
// ===== library types =====

TYPE "udtError_MQTT"
   STRUCT
      ConSendErr : Bool;   // Connect send error
      ConSendTO : Bool;   // Connect send timeout
      ConAckRcvErr : Bool;   // Connack receive error
      ConAckTO : Bool;   // Connack timeout
      ConAckIncReply : Bool;   // Conack incorrect reply (header)
      ConAckIncLen : Bool;   // Conack incorrect remaining length
      ConAckUnacProt : Bool;   // Conack unacceptable protocol version (0x01)
      ConAckIdRej : Bool;   // Conack ID rejected (0x02)
      ConAckSerUn : Bool;   // Conack server unavailable (0x03)
      ConAckUserPass : Bool;   // Conack incorerct user/password (0x04)
      ConAckNotAut : Bool;   // Conack not authorized (0x05)
      ConAckUnknown : Bool;   // Conack unknow erro code (>0x05)
      PubSendErr : Bool;   // Publish send error
      PubSendTO : Bool;   // Publish send timeout
      PubAckRcvErr : Bool;   // Puback receive error
      PubAckTO : Bool;   // Puback receive timeout
      PubAckIncReply : Bool;   // Puback incorerct reply (header)
      PubAckIncLen : Bool;   // Puback incorrect remaining length
      PubAckPacketID : Bool;   // Puback incorrect Packet ID
      SubSendErr : Bool;   // Subscribe send error
      SubSendTimeout : Bool;   // Subscribe send timeout
      SubAckIncReply : Bool;   // Suback incorrect reply
      SubAckPacketID : Bool;   // Suback incorrect Packet ID
      SubAckRcvErr : Bool;   // Suback receive error
      SubAckTO : Bool;   // Suback receive timeout
      SubTopicNotFound : Bool;   // Message sent to PLC, but not subscribed to topic
      SubSendPubAckErr : Bool;   // Error sending pub ack message
      SubSendPubAckTO : Bool;   // Send pub ack timeout
      TcpErr : Bool;   // TCP connection failed
      TcpTO : Bool;   // TCP connection timeout
      QueueOverflow : Bool;   // Queue overlow
   END_STRUCT;
END_TYPE

TYPE "udtMQTT_PublishMessage"
   STRUCT
      iStatus : Int;   // 0 - Disabled,10 - Ready to Send
      iQoS : Int;
      sTopic : String;
      byValue : Array[0..100] of Byte;
      iMessageLength : DInt;
   END_STRUCT;
END_TYPE

TYPE "udtMQTT_PublishMessageBuffer"
   STRUCT
      iIndexWrite : Int;
      iIndexMax : Int := 50;
      bErrorOverfill : Bool;
      Message : Array[1..10] of "udtMQTT_PublishMessage";
   END_STRUCT;
END_TYPE

TYPE "udtMQTT_SubscribeMessage"
   STRUCT
      iStatus : Int;   // 0 - Disabled, 10 - Ready to subscribe, 20 - subscribed, 30 - New data
      iQoS : Int;
      sTopic : String[75];
      byValue : Array[0..75] of Byte;
      iMessageLength : Int;
   END_STRUCT;
END_TYPE

TYPE "udtMQTT_SubcribeMessageBuffer"
   STRUCT
      Message : Array[1..20] of "udtMQTT_SubscribeMessage";
   END_STRUCT;
END_TYPE

FUNCTION_BLOCK "fbMQTT_V2"   // FB19, SCL
{ S7_Optimized_Access := 'TRUE' }
VERSION : 0.1
   VAR_INPUT
      sInClientID : String;   // Client ID, 23 char max
      sInUserName : String;
      sInPassword : String;
      bInCleanSession : Bool;   // 0=Reuse prev session; 1=Discard prev sessions and start new one
      bInResetError : Bool;
   END_VAR
   VAR_OUTPUT
      bOutError : Bool;
   END_VAR
   VAR_IN_OUT
      ERROR_MQTT : "udtError_MQTT";
      TCON_Param : TCON_Param;
   END_VAR
   VAR
      iStatePublish : Int;
      iStateSubscribe : Int;
      iStateTCP_Receive : Int;
      iSelQueueIndexPublish : Int;
      iPublishIndex : Int;
      uiSendLen : UInt;
      udiReceiveLen : UDInt;
      uiPubPacketID : UInt;
      bPubInProgress : Bool;
      iSubscribeIndex : Int;
      uiSubPacketID : UInt;
      iSubMessageIndex : Int;
      bSubInProgress : Bool;
      bSubReceiveInProgress : Bool;
      iSubReceivedQoS : Int;
      iReceivedTopicLength : Int;
      sReceivedTopic : String;
      iTopicIndex : Int;
      bConAckReceived : Bool;
      bPubAckReceived : Bool;
      bSubAckReceived : Bool;
      bPublishReceived : Bool;
      iPayloadStartIndex : Int;
      iEndOfPayloadIndex : Int;
      byData : Array[1..200] of Byte;   // Max: id+user+password+buffer
      byDataNewMessage : Array[1..300] of Byte;
      fbTCON : TCON;
      fbTDISCON : TDISCON;
      fbTSEND : TSEND;
      fbTRCV : TRCV;
      TON_TimeoutPub : TON_TIME;
      TON_TimeoutSub : TON_TIME;
      TON_ReceiveDataComplete : TON_TIME;
      TON_DelaySubscribe : TON_TIME;   // To space out traffic, wait 5 seconds after MQTT connection to subscribe
      iNewDataIndex : Int := 1;
      bNewDataReceived : Bool;
      bTCP_Connected : Bool;
      bMQTT_Connected : Bool;
      iLen : Int;
      iStatePrevPub : Int;
      bStateTransitionPub : Bool;
      udiSetReceiveLen : UDInt;
      wTemp : Word;
      wTemp2 : Word;
      wTemp3 : Word;
      wTemp4 : Word;
      byMSB : Byte;
      byLSB : Byte;
      iStatePrevSub : Int;
      bStateTransitionSub : Bool;
      bReceiveMessageComplete : Bool;
      iReceiveMessageLength : Int;
      iReceiveLengthCalcIndex : Int;
      iErrIndex : Int := 1;
   END_VAR
   VAR_TEMP
      i : Int;
      j : Int;
      iStartingIndex : Int;
      iTemp : Int;
      byTemp : Byte;
      uiTemp : UInt;
      uiTopicLen : UInt;
      multiplier : Int;
      byTopic : Array[1..500] of Byte;
      byReceivedPayload : Array[1..500] of Byte;
      iLowerByte : Int;
      iHigherByte : Int;
      sSearchString : String;
      bTopicNotFound : Bool;
   END_VAR
   VAR CONSTANT
      ciPublishQueueSize : Int := 10;
      ciPubIdle : Int := 10;
      ciPubError : Int := 999;
      ciEstablishTCP : Int := 100;
      ciPubConnect : Int := 20;
      ciPubConnectSend : Int := 30;
      ciPubWaitConnack : Int := 40;
      ciPubPublish : Int := 50;
      ciPubSend : Int := 60;
      ciPubWaitPubAck : Int := 70;
      ciPubRestart : Int := -1;
      ciSubQueueSize : Int := 20;
      ciSubIdle : Int := 10;
      ciSubError : Int := 999;
      ciSubWaitTCP : Int := 20;
      ciSubSubscribe : Int := 30;
      ciSubSendSubscribe : Int := 40;
      ciSubWaitSuback : Int := 50;
      ciSubDataReceived : Int := 60;
      ciSubSendPubAck : Int := 70;
      ciRecIdle : Int := 10;
      ciRecDataReceived : Int := 20;
      ciRecParseData : Int := 30;
      ciRecConAck : Int := 40;
      ciRecPubAck : Int := 50;
      ciRecSubAck : Int := 60;
      ciRecPubReceived : Int := 70;
   END_VAR
BEGIN
   //Publish state machine
   //Test comment
   #iStatePrevPub := #iStatePublish;
   CASE #iStatePublish OF
       #ciPubIdle:
           // Update max queue index
           "dbMQTT_MessageBuffer".OutgoingMessages.iIndexMax := #ciPublishQueueSize;

           //connect by default
           IF NOT #bTCP_Connected THEN
               #iStatePublish := #ciEstablishTCP;
           END_IF;

           IF #bTCP_Connected AND NOT #bMQTT_Connected THEN
               #iStatePublish := #ciPubConnect;
           END_IF;


           // Already select element to send?
           IF #iSelQueueIndexPublish > 0 THEN
               IF #bTCP_Connected AND #bMQTT_Connected AND #iStateSubscribe = #ciSubIdle THEN
                   //Only publish if subscribe state machine is also idle
                   #iStatePublish := #ciPubPublish;
               END_IF;
           ELSE
               // Find element in the queue to send
               FOR #i := 1 TO "dbMQTT_MessageBuffer".OutgoingMessages.iIndexMax DO
                   // Check if element is ready in the queue
                   IF ("dbMQTT_MessageBuffer".OutgoingMessages.Message[#i].iStatus = "ciReadyToPublish") THEN
                       #iSelQueueIndexPublish := #i;
                       EXIT;
                   END_IF;
               END_FOR;
           END_IF;

       #ciPubConnect: // Send connect message
           ////////////////////////////////////
           // Create connect message
           ////////////////////////////////////

           //********* Configure Fixed Header ***********//
           #iPublishIndex := 1;
           #byData[#iPublishIndex] := 2#00010000;   // Packet type 0x1; Flags 0x0 (reserved)
           #iPublishIndex := #iPublishIndex + 1;

           //Reset all subscriptions
           FOR #i := 1 TO 20 BY 1 DO
               "dbMQTT_MessageBuffer".IncomingMessages.Message[#i].iStatus := "ciSubDisabled";
           END_FOR;

           // Calculate remaining length (see MQTT doc)
           #iLen := 12 + LEN(#sInClientID);
           IF LEN(#sInUserName) > 0 THEN
               #iLen := #iLen + LEN(#sInUserName) + 2;
           END_IF;
           IF LEN(#sInPassword) > 0 THEN
               #iLen := #iLen + LEN(#sInPassword) + 2;
           END_IF;
           REPEAT
               #byTemp := INT_TO_BYTE(#iLen MOD 128);
               #iLen := #iLen / 128;
               // if there are more data to encode, set the top bit of this byte 286
               IF #iLen > 0 THEN
                   #byTemp := #byTemp OR 128;
               END_IF;
               #byData[#iPublishIndex] := #byTemp;
               #iPublishIndex := #iPublishIndex + 1;
           UNTIL #iLen <= 0 END_REPEAT;

           //********* Variable Header ***********//
           #byData[#iPublishIndex] := 16#00;    // Length MSB
           #iPublishIndex := #iPublishIndex + 1;
           #byData[#iPublishIndex] := 16#04;    // Length LSB
           #iPublishIndex := #iPublishIndex + 1;
           #byData[#iPublishIndex] := CHAR_TO_BYTE('M');
           #iPublishIndex := #iPublishIndex + 1;
           #byData[#iPublishIndex] := CHAR_TO_BYTE('Q');
           #iPublishIndex := #iPublishIndex + 1;
           #byData[#iPublishIndex] := CHAR_TO_BYTE('T');
           #iPublishIndex := #iPublishIndex + 1;
           #byData[#iPublishIndex] := CHAR_TO_BYTE('T');
           #iPublishIndex := #iPublishIndex + 1;
           #byData[#iPublishIndex] := 16#04;     // Protocol level 0x04
           #iPublishIndex := #iPublishIndex + 1;

           // Build connect flags, ignoring will message
           #byData[#iPublishIndex] := 16#00;
           IF LEN(#sInUserName) > 0 THEN
               #byData[#iPublishIndex] := #byData[#iPublishIndex] OR 2#10000000;
           END_IF;
           IF LEN(#sInPassword) > 0 THEN
               #byData[#iPublishIndex] := #byData[#iPublishIndex] OR 2#01000000;
           END_IF;
           IF #bInCleanSession THEN
               #byData[#iPublishIndex] := #byData[#iPublishIndex] OR 2#00000010;
           END_IF;
           #iPublishIndex := #iPublishIndex + 1;
           #byData[#iPublishIndex] := 16#0E;  // Keepalive MSB, in seconds
           #iPublishIndex := #iPublishIndex + 1;
           #byData[#iPublishIndex] := 16#10;  // Keepalive LSB, in seconds
           #iPublishIndex := #iPublishIndex + 1;

           // Payload - client ID
           #iLen := LEN(#sInClientID);
           #byData[#iPublishIndex] := WORD_TO_BYTE(SHR(IN := INT_TO_WORD(#iLen), N := 8));   // String lenght MSB
           #iPublishIndex := #iPublishIndex + 1;
           #byData[#iPublishIndex] := WORD_TO_BYTE(INT_TO_WORD(#iLen) AND 16#00FF);   // String lenght LSB            
           #iPublishIndex := #iPublishIndex + 1;
           FOR #i := 1 TO #iLen DO
               #byData[#iPublishIndex] := CHAR_TO_BYTE(#sInClientID[#i]);
               #iPublishIndex := #iPublishIndex + 1;
           END_FOR;

           // Payload - User name
           IF LEN(#sInUserName) > 0 THEN
               #iLen := LEN(#sInUserName);
               #byData[#iPublishIndex] := WORD_TO_BYTE(SHR(IN := INT_TO_WORD(#iLen), N := 8));   // String lenght MSB
               #iPublishIndex := #iPublishIndex + 1;
               #byData[#iPublishIndex] := WORD_TO_BYTE(INT_TO_WORD(#iLen) AND 16#00FF);   // String lenght LSB            
               #iPublishIndex := #iPublishIndex + 1;
               FOR #i := 1 TO #iLen DO
                   #byData[#iPublishIndex] := CHAR_TO_BYTE(#sInUserName[#i]);
                   #iPublishIndex := #iPublishIndex + 1;
               END_FOR;
           END_IF;

           // Payload - password
           IF LEN(#sInPassword) > 0 THEN
               #iLen := LEN(#sInPassword);
               #byData[#iPublishIndex] := WORD_TO_BYTE(SHR(IN := INT_TO_WORD(#iLen), N := 8));   // String lenght MSB
               #iPublishIndex := #iPublishIndex + 1;
               #byData[#iPublishIndex] := WORD_TO_BYTE(INT_TO_WORD(#iLen) AND 16#00FF);   // String lenght LSB            
               #iPublishIndex := #iPublishIndex + 1;
               FOR #i := 1 TO #iLen DO
                   #byData[#iPublishIndex] := CHAR_TO_BYTE(#sInPassword[#i]);
                   #iPublishIndex := #iPublishIndex + 1;
               END_FOR;
           END_IF;

           //********* Send Packet ***********//
           #uiSendLen := INT_TO_UINT(#iPublishIndex - 1);   // Update packet length
           #iStatePublish := #ciPubConnectSend;  // Send packet packet

       #ciPubConnectSend:
           IF #fbTSEND.DONE THEN
               // All good. Receive conack message
               // We know exactly the conack message size
               #udiReceiveLen := 4;
               #iStatePublish := #ciPubWaitConnack;
           ELSIF #fbTSEND.ERROR THEN
               // Sending error
               #ERROR_MQTT.ConSendErr := true;
               #iStatePublish := #ciPubError;
           ELSIF #TON_TimeoutPub.Q THEN
               #ERROR_MQTT.ConSendTO := true;
               #iStatePublish := #ciPubError;
           END_IF;

       #ciPubWaitConnack:
           IF #bConAckReceived THEN
               //Reset received flag
               #bConAckReceived := FALSE;
               // Parse received data
               // We know that we got an expected length
               // Header should be 0x20
               IF #byDataNewMessage[1] <> 16#20 THEN
                   #ERROR_MQTT.ConAckIncReply := true;
                   #iStatePublish := #ciPubError;
                   // Remaining lenght should be 2
               ELSIF #byDataNewMessage[2] <> 2 THEN
                   #ERROR_MQTT.ConAckIncLen := true;
                   #iStatePublish := #ciPubError;
                   // TODO: Parse SP flag?
                   // Return code should be 0    
               ELSIF #byDataNewMessage[4] <> 0 THEN
                   // Parse error code
                   IF #byDataNewMessage[4] = 1 THEN
                       #ERROR_MQTT.ConAckUnacProt := TRUE;
                   ELSIF #byDataNewMessage[4] = 2 THEN
                       #ERROR_MQTT.ConAckIdRej := TRUE;
                   ELSIF #byDataNewMessage[4] = 3 THEN
                       #ERROR_MQTT.ConAckSerUn := TRUE;
                   ELSIF #byDataNewMessage[4] = 4 THEN
                       #ERROR_MQTT.ConAckUserPass := TRUE;
                   ELSIF #byDataNewMessage[4] = 5 THEN
                       #ERROR_MQTT.ConAckNotAut := TRUE;
                   ELSE
                       #ERROR_MQTT.ConAckUnknown := TRUE;
                   END_IF;
                   #iStatePublish := #ciPubError;
               ELSE
                   // All good
                   #bMQTT_Connected := true;
                   #iStatePublish := #ciPubIdle;
               END_IF;
           (*ELSIF #fbTRCV.ERROR THEN
               // Receive error
               #ERROR_MQTT.ConAckRcvErr := true;
               "dbTestingJJC".wDisError := #fbTRCV.STATUS;
               #iStatePublish := #ciPubError;*)
           ELSIF #TON_TimeoutPub.Q THEN
               #ERROR_MQTT.ConAckTO := true;
               #iStatePublish := #ciPubError;
           END_IF;

       #ciPubPublish:
           ////////////////////////////////////
           // Create publish message
           ////////////////////////////////////

           //********* Configure Fixed Header ***********//
           #iPublishIndex := 1;
           #byData[#iPublishIndex] := 2#00110000;   // Packet type 0x3;
           IF #bPubInProgress THEN
               #byData[#iPublishIndex] := #byData[#iPublishIndex] OR 2#00001000; // DUP flag. Re-delivery attempt
           ELSE
               // New send attempt - Increment Packet ID
               #uiPubPacketID := #uiPubPacketID + 1;
           END_IF;
           // QoS flag, assuming 0 by default
           IF "dbMQTT_MessageBuffer".OutgoingMessages.Message[#iSelQueueIndexPublish].iQoS = 1 THEN
               #byData[#iPublishIndex] := #byData[#iPublishIndex] OR 2#00000010; // QoS flag
           END_IF;
           //TODO: QoS 2 is not currently implemented by adafruit
           // TODO: Ignoring retain flag for now
           #iPublishIndex := #iPublishIndex + 1;

           // Calculate remaining length (see MQTT doc)
           // No lenght for the payload
           #iLen := LEN("dbMQTT_MessageBuffer".OutgoingMessages.Message[#iSelQueueIndexPublish].sTopic) + 2 + DINT_TO_INT("dbMQTT_MessageBuffer".OutgoingMessages.Message[#iSelQueueIndexPublish].iMessageLength);
           IF "dbMQTT_MessageBuffer".OutgoingMessages.Message[#iSelQueueIndexPublish].iQoS > 0 THEN
               // Adding packet ID for QoS 1 and 2
               #iLen := #iLen + 2;
           END_IF;
           REPEAT
               #byTemp := INT_TO_BYTE(#iLen MOD 128);
               #iLen := #iLen / 128;
               // if there are more data to encode, set the top bit of this byte 286
               IF #iLen > 0 THEN
                   #byTemp := #byTemp OR 128;
               END_IF;
               #byData[#iPublishIndex] := #byTemp;
               #iPublishIndex := #iPublishIndex + 1;
           UNTIL #iLen <= 0 END_REPEAT;

           //********* Variable Header ***********//
           // Topic name
           #iLen := LEN("dbMQTT_MessageBuffer".OutgoingMessages.Message[#iSelQueueIndexPublish].sTopic);
           #byData[#iPublishIndex] := WORD_TO_BYTE(SHR(IN := INT_TO_WORD(#iLen), N := 8));   // String lenght MSB
           #iPublishIndex := #iPublishIndex + 1;
           #byData[#iPublishIndex] := WORD_TO_BYTE(INT_TO_WORD(#iLen) AND 16#00FF);   // String lenght LSB
           #iPublishIndex := #iPublishIndex + 1;
           FOR #i := 1 TO #iLen DO
               #byData[#iPublishIndex] := CHAR_TO_BYTE("dbMQTT_MessageBuffer".OutgoingMessages.Message[#iSelQueueIndexPublish].sTopic[#i]);
               #iPublishIndex := #iPublishIndex + 1;
           END_FOR;
           // packet ID
           IF "dbMQTT_MessageBuffer".OutgoingMessages.Message[#iSelQueueIndexPublish].iQoS > 0 THEN
               #byData[#iPublishIndex] := WORD_TO_BYTE(SHR(IN := UINT_TO_WORD(#uiPubPacketID), N := 8));   // Packet ID MSB
               #iPublishIndex := #iPublishIndex + 1;
               #byData[#iPublishIndex] := WORD_TO_BYTE(UINT_TO_WORD(#uiPubPacketID) AND 16#00FF);   // PacketID LSB
               #iPublishIndex := #iPublishIndex + 1;
           END_IF;

           //********* Payload ***********//
           // The exact data format is not defined in the MQTT spec
           // Assuming strings, without string length
           // According to the spec, server should calcualte the lenght of the payload
           #iLen := DINT_TO_INT("dbMQTT_MessageBuffer".OutgoingMessages.Message[#iSelQueueIndexPublish].iMessageLength);
           FOR #i := 0 TO #iLen - 1 DO
               #byData[#iPublishIndex] := "dbMQTT_MessageBuffer".OutgoingMessages.Message[#iSelQueueIndexPublish].byValue[#i];
               #iPublishIndex := #iPublishIndex + 1;
           END_FOR;

           // Send message
           #bPubInProgress := true;
           #uiSendLen := INT_TO_UINT(#iPublishIndex - 1);   // Update packet length
           #iStatePublish := #ciPubSend;

       #ciPubSend:
           IF #fbTSEND.DONE THEN
               // QoS=1: Should receive puback message
               IF "dbMQTT_MessageBuffer".OutgoingMessages.Message[#iSelQueueIndexPublish].iQoS = 1 THEN
                   #udiReceiveLen := 4;    // Wes should receive exactly 4 bytes
                   #iStatePublish := #ciPubWaitPubAck;
               ELSE
                   // QoS=0; No response from the server
                   // Remove message from the queue
                   "dbMQTT_MessageBuffer".OutgoingMessages.Message[#iSelQueueIndexPublish].iStatus := "ciDisablePublish";
                   #iSelQueueIndexPublish := 0;
                   #bPubInProgress := false;
                   #iStatePublish := #ciPubIdle;
               END_IF;
               // TODO: Handle QoS 2?
           ELSIF #fbTSEND.ERROR THEN
               // Send error
               #ERROR_MQTT.PubSendErr := true;
               #iStatePublish := #ciPubError;
           ELSIF #TON_TimeoutPub.Q THEN
               #ERROR_MQTT.PubSendTO := true;
               #iStatePublish := #ciPubError;
           END_IF;

       #ciEstablishTCP:
           // Wait for done or error flag
           IF #fbTCON.DONE THEN
               // TCP connection established 
               #bTCP_Connected := true;
               #bMQTT_Connected := false;
               #iStatePublish := #ciPubConnect;
           ELSIF #fbTCON.ERROR THEN
               // Connection failed
               #ERROR_MQTT.TcpErr := true;
               IF #fbTCON.STATUS = 16#80A3 THEN
                   #TCON_Param.ID := #TCON_Param.ID + 1;
               END_IF;
               IF #TCON_Param.ID > 9 THEN
                   #TCON_Param.ID := 1;
               END_IF;
               #iStatePublish := #ciPubError;
           ELSIF #TON_TimeoutPub.Q THEN
               #ERROR_MQTT.TcpTO := true;
               #iStatePublish := #ciPubError;
           END_IF;

       #ciPubWaitPubAck:
           IF #bPubAckReceived THEN
               #bPubAckReceived := false;
               // Parse received data
               // We know that we got an expected length
               // Header should be 0x40
               IF #byDataNewMessage[2] <> 16#02 THEN
                   // Wrong pub ack remaining lenght
                   // TODO pub ack length error
                   #iStatePublish := #ciPubError;
               ELSE
                   // Variable header = message id
                   #uiTemp := WORD_TO_UINT(SHL(IN := BYTE_TO_WORD(#byDataNewMessage[3]), N := 8) + BYTE_TO_WORD(#byDataNewMessage[4]));
                   IF #uiTemp <> #uiPubPacketID THEN
                       // Incorerct packet ID
                       #ERROR_MQTT.PubAckPacketID := TRUE;
                       #iStatePublish := #ciPubError;
                   ELSE
                       // All good. Reset queue and restart
                       "dbMQTT_MessageBuffer".OutgoingMessages.Message[#iSelQueueIndexPublish].iStatus := "ciDisablePublish";
                       #iSelQueueIndexPublish := 0;
                       #bPubInProgress := false;
                       #iStatePublish := #ciPubIdle;
                   END_IF;
               END_IF;
           ELSIF #fbTRCV.ERROR THEN
               // Receive error
               #ERROR_MQTT.PubAckRcvErr := TRUE;
               #iStatePublish := #ciPubError;
           ELSIF #TON_TimeoutPub.Q THEN
               #ERROR_MQTT.PubAckTO := true;
               #iStatePublish := #ciPubError;
           END_IF;

       #ciPubError:
           // Reset TCP connection
           #bMQTT_Connected := false;
           #bTCP_Connected := false;
           IF #fbTDISCON.DONE THEN
               #iStatePublish := #ciPubRestart;
           ELSIF #TON_TimeoutPub.Q THEN
               // Already wait for timeout, just jump to idle
               #iStatePublish := #ciPubIdle;
               #iNewDataIndex := 1;
           END_IF;

       #ciPubRestart:
           // Wait before restarting after the error
           IF #TON_TimeoutPub.Q THEN
               // Restart from IDLE
               #iStatePublish := #ciPubIdle;
               #iNewDataIndex := 1;
           END_IF;

       ELSE
           #iStatePublish := #ciPubIdle;

   END_CASE;

   // Timeoout timer
   #bStateTransitionPub := #iStatePublish <> #iStatePrevPub;
   #TON_TimeoutPub(IN := ((NOT #bStateTransitionPub) AND (#iStatePublish <> #ciPubIdle) AND #iStateSubscribe = #ciSubIdle), PT := T#20S);

   //subscribe state machine
   #iStatePrevSub := #iStateSubscribe;
   CASE #iStateSubscribe OF
       #ciSubIdle:
           #bSubInProgress := false;
           #bSubReceiveInProgress := false;
           //Wait until TCP and MQTT connected and publish is idle
           IF #TON_DelaySubscribe.Q AND #iStatePublish = #ciPubIdle  THEN
               //check if any new data has arrived
               IF #bPublishReceived THEN
                   //Reset flag
                   #bPublishReceived := false;
                   //if data has arrived, move to data received state
                   #iStateSubscribe := #ciSubDataReceived;
                   //Set flag to prevent sending other messages out
                   #bSubReceiveInProgress := true;
               END_IF;

               //check for any unsubscribed topics
               IF NOT #bSubReceiveInProgress THEN
                   FOR #i := 1 TO #ciSubQueueSize BY 1 DO
                       IF "dbMQTT_MessageBuffer".IncomingMessages.Message[#i].iStatus = "ciSubReadyToSub" THEN
                           //If unsubscribed topic found, move to sub state and stop looking for new topics
                           #iStateSubscribe := #ciSubSubscribe;
                           #iSubscribeIndex := #i;
                           #bSubInProgress := TRUE;
                           EXIT;
                       END_IF;
                   END_FOR;
               END_IF;
           END_IF;

       #ciSubSubscribe:
           //create subscribe MQTT packet
           #i := 1;
           #iSubMessageIndex := 1;
           #byData[#iSubMessageIndex] := 2#10000010;   // Packet type 0x8; Flags 0x0 (reserved)
           #iSubMessageIndex := #iSubMessageIndex + 1;

           // Calculate remaining length (see MQTT doc)
           // packet identifier (2) + topic length (2) + length of topic + QoS (1)
           #iLen := LEN("dbMQTT_MessageBuffer".IncomingMessages.Message[#iSubscribeIndex].sTopic) + 5;
           //Create encoding for packet length
           REPEAT
               #byTemp := INT_TO_BYTE(#iLen MOD 128);
               #iLen := #iLen / 128;
               // if there are more data to encode, set the top bit of this byte 286
               IF #iLen > 0 THEN
                   #byTemp := #byTemp OR 128;
               END_IF;
               #byData[#iSubMessageIndex] := #byTemp;
               #iSubMessageIndex := #iSubMessageIndex + 1;
           UNTIL #iLen <= 0 END_REPEAT;
           //increment packet ID and encode into variable header
           #uiSubPacketID := #uiSubPacketID + 1;
           #byData[#iSubMessageIndex] := WORD_TO_BYTE(SHR(IN := UINT_TO_WORD(#uiSubPacketID), N := 8));   // Packet ID MSB
           #iSubMessageIndex := #iSubMessageIndex + 1;
           #byData[#iSubMessageIndex] := WORD_TO_BYTE(UINT_TO_WORD(#uiSubPacketID) AND 16#00FF);   // PacketID LSB
           #iSubMessageIndex := #iSubMessageIndex + 1;

           //build payload
           //Only 1 topic. 2 bytes for length, topic, 1 byte for QoS
           //Length
           #uiTopicLen := INT_TO_UINT(LEN("dbMQTT_MessageBuffer".IncomingMessages.Message[#iSubscribeIndex].sTopic));
           #byData[#iSubMessageIndex] := WORD_TO_BYTE(SHR(IN := UINT_TO_WORD(#uiTopicLen), N := 8));   // Packet ID MSB
           #iSubMessageIndex := #iSubMessageIndex + 1;
           #byData[#iSubMessageIndex] := WORD_TO_BYTE(UINT_TO_WORD(#uiTopicLen) AND 16#00FF);   // PacketID LSB
           #iSubMessageIndex := #iSubMessageIndex + 1;
           // Topic name
           #iLen := LEN("dbMQTT_MessageBuffer".IncomingMessages.Message[#iSubscribeIndex].sTopic);
           FOR #i := 1 TO #iLen DO
               #byData[#iSubMessageIndex] := CHAR_TO_BYTE("dbMQTT_MessageBuffer".IncomingMessages.Message[#iSubscribeIndex].sTopic[#i]);
               #iSubMessageIndex := #iSubMessageIndex + 1;

           END_FOR;
           //QoS
           IF "dbMQTT_MessageBuffer".IncomingMessages.Message[#iSubscribeIndex].iQoS = 1 THEN
               #byData[#iSubMessageIndex] := 2#00000001;
           ELSE
               #byData[#iSubMessageIndex] := 2#00000000;
           END_IF;
           #uiSendLen := INT_TO_UINT(#iSubMessageIndex);
           #iStateSubscribe := #ciSubSendSubscribe;

       #ciSubSendSubscribe:
           IF #fbTSEND.DONE THEN

               #iStateSubscribe := #ciSubWaitSuback;
               IF "dbMQTT_MessageBuffer".IncomingMessages.Message[#iSubscribeIndex].iQoS = 0 THEN
                   #udiReceiveLen := 5;    // Wes should receive exactly 4 bytes
                   #iStateSubscribe := #ciSubWaitSuback;
               END_IF;
           ELSIF #fbTSEND.ERROR THEN
               // Send error
               #ERROR_MQTT.PubSendErr := true;
               #iStateSubscribe := #ciPubError;
           ELSIF #TON_TimeoutSub.Q THEN
               #ERROR_MQTT.PubSendTO := true;
               #iStateSubscribe := #ciPubError;
           END_IF;

       #ciSubWaitSuback:
           //validate packet received. Should have same packet ID
           //
           IF #bSubAckReceived THEN
               #bSubAckReceived := false;
               // Parse received data
               // We know that we got an expected length
               // Header should be 0x40

               // Variable header = message id
               #uiTemp := WORD_TO_UINT(SHL(IN := BYTE_TO_WORD(#byDataNewMessage[3]), N := 8) + BYTE_TO_WORD(#byDataNewMessage[4]));

               IF #uiTemp <> #uiSubPacketID THEN
                   // Incorerct packet ID
                   #ERROR_MQTT.SubAckPacketID := TRUE;
                   #iStateSubscribe := #ciSubError;
                   //TODO also check QoS?
               ELSE
                   // All good. Reset queue and restart

                   "dbMQTT_MessageBuffer".IncomingMessages.Message[#iSubscribeIndex].iStatus := "ciSubSubscribed";
                   #iStateSubscribe := #ciSubIdle;
               END_IF;
           (* ELSIF #fbTRCV.ERROR THEN
               // Receive error
               #ERROR_MQTT.SubAckRcvErr := TRUE;
               #iStateSubscribe := #ciSubError; *)
           ELSIF #TON_TimeoutSub.Q THEN
               #ERROR_MQTT.SubAckTO := true;
               #iStateSubscribe := #ciSubError;
           END_IF;


       #ciSubDataReceived:
           //reset flag
           #bSubReceiveInProgress := false;
           //find QoS
           #iSubMessageIndex := 1;
           #iSubReceivedQoS := 0;
           //TODO handling for QoS 2
           IF (#byDataNewMessage[#iSubMessageIndex] AND 2#00000010) = 2#00000010 THEN
               #iSubReceivedQoS := 1;
           END_IF;

           //calculate message length
           #multiplier := 1;
           #iLen := 0;
           #iSubMessageIndex := 2;
           REPEAT

               #byTemp := #byDataNewMessage[#iSubMessageIndex];
               #iLen := #iLen + (#byTemp AND 127) * #multiplier;
               #multiplier := #multiplier * 128;
               //TODO implement exception for length error

               #iSubMessageIndex := #iSubMessageIndex + 1;
           UNTIL ((#byTemp AND 128) = 0) END_REPEAT;

           //find end index of message
           #iEndOfPayloadIndex := #iLen + #iSubMessageIndex - 1;

           //find topic name
           //find topic length
           #wTemp := 16#0000;
           #wTemp2 := 16#0000;
           #wTemp := #wTemp OR #byDataNewMessage[#iSubMessageIndex];
           #iSubMessageIndex := #iSubMessageIndex + 1;
           #wTemp2 := #byDataNewMessage[#iSubMessageIndex];
           #wTemp3 := SHL(IN := #wTemp, N := 8);
           #wTemp4 := #wTemp OR #wTemp2;
           #iReceivedTopicLength := WORD_TO_INT(IN := #wTemp4);
           #iSubMessageIndex := #iSubMessageIndex + 1;
           #iStartingIndex := #iSubMessageIndex;
           #j := 1;
           FOR #i := #iStartingIndex TO #iStartingIndex + #iReceivedTopicLength BY 1 DO
               #byTopic[#j] := #byDataNewMessage[#iSubMessageIndex];
               #j := #j + 1;
               #iSubMessageIndex := #iSubMessageIndex + 1;
           END_FOR;

           Chars_TO_Strg(Chars:=#byTopic, pChars:=0, Cnt:=INT_TO_UINT(#iReceivedTopicLength), Strg=>#sReceivedTopic);
           //find index of topic
           #bTopicNotFound := TRUE;
           FOR #i := 1 TO #ciSubQueueSize BY 1 DO

               IF ("dbMQTT_MessageBuffer".IncomingMessages.Message[#i].sTopic = #sReceivedTopic) THEN
                   #iTopicIndex := #i;
                   #bTopicNotFound := FALSE;
                   EXIT;
               END_IF;
           END_FOR;

           //Throw error if topic not found
           IF #bTopicNotFound THEN
               #ERROR_MQTT.SubTopicNotFound := TRUE;
               #iStatePrevSub := #ciSubError;
           END_IF;

           //Depending on QoS go to idle or send PubAck reply
           IF (#iSubReceivedQoS = 0) THEN
               #iStateSubscribe := #ciSubIdle;
           ELSIF (#iSubReceivedQoS = 1) THEN

               //Find packet ID
               #byLSB := #byDataNewMessage[#iSubMessageIndex];
               #iSubMessageIndex := #iSubMessageIndex + 1;
               #byMSB := #byDataNewMessage[#iSubMessageIndex];

               //build reply message
               //Control packet 16#40
               #byData[1] := 16#40;
               //remaining length is 2
               #byData[2] := 16#02;
               //add packet id
               #byData[3] := #byMSB;
               #byData[4] := #byLSB;
               #uiSendLen := 4;

               #iStateSubscribe := #ciSubSendPubAck;
           END_IF;

           //get message
           IF NOT #bTopicNotFound THEN
               #iPayloadStartIndex := #iSubMessageIndex;
               #j := 0;
               FOR #i := #iPayloadStartIndex - 1 TO #iEndOfPayloadIndex BY 1 DO

                   "dbMQTT_MessageBuffer".IncomingMessages.Message[#iTopicIndex].byValue[#j] := #byDataNewMessage[#i];
                   #j := #j + 1;
               END_FOR;



               //move topic and payload into received queue and set status

               "dbMQTT_MessageBuffer".IncomingMessages.Message[#iTopicIndex].iStatus := "ciSubMessageReceived";
               "dbMQTT_MessageBuffer".IncomingMessages.Message[#iTopicIndex].iMessageLength := #j;


           END_IF;

       #ciSubSendPubAck:
           IF #fbTSEND.DONE THEN
               #iStateSubscribe := #ciSubIdle;
           ELSIF #fbTSEND.ERROR THEN
               // Send error
               #ERROR_MQTT.SubSendPubAckErr := true;
               #iStateSubscribe := #ciPubError;
           ELSIF #TON_TimeoutSub.Q THEN
               #ERROR_MQTT.SubSendPubAckTO := true;
               #iStateSubscribe := #ciPubError;
           END_IF;

       #ciSubError:
           // Reset TCP connection
           #bMQTT_Connected := false;
           #bTCP_Connected := false;
           IF #fbTDISCON.DONE OR #fbTDISCON.ERROR THEN
               #iStateSubscribe := #ciPubRestart;
           ELSIF #TON_TimeoutSub.Q THEN
               // Already wait for timeout, just jump to idle
               #iStateSubscribe := #ciSubIdle;
           END_IF;

       #ciPubRestart:
           // Wait before restarting after the error
           IF #TON_TimeoutSub.Q THEN
               // Restart from IDLE
               #iStateSubscribe := #ciSubIdle;
           END_IF;


       ELSE
           #iStateSubscribe := #ciSubIdle;

   END_CASE;

   // Timeoout timer
   #bStateTransitionSub := #iStateSubscribe <> #iStatePrevSub;
   #TON_TimeoutSub(IN := ((NOT #bStateTransitionSub) AND (#iStateSubscribe <> #ciSubIdle)),
                   PT := T#20S);

   #TON_DelaySubscribe(IN := #bMQTT_Connected,
                       PT := T#3S);


   //Receive TCP data AND set flags
   IF #bReceiveMessageComplete AND #iNewDataIndex > 0 THEN

       IF #byDataNewMessage[1] = 16#20 THEN
           #bConAckReceived := TRUE;
       END_IF;

       IF #byDataNewMessage[1] = 16#40 THEN
           #bPubAckReceived := TRUE;
       END_IF;

       IF #byDataNewMessage[1] = 16#90 THEN
           #bSubAckReceived := TRUE;
       END_IF;

       IF (#byDataNewMessage[1] AND 2#11110000) = 16#30 AND #iStateSubscribe = #ciSubIdle THEN
           #bPublishReceived := TRUE;
       END_IF;

       #iNewDataIndex := 1;

       #bReceiveMessageComplete := FALSE;
       #iReceiveMessageLength := 0;


   END_IF;



   //**********************************************************************************************************************
   // Communicaiton FBs

   //Monitor TCP connection, if receive error has error above 80A1, then a comm error has occured and connection should be re-established
   IF #fbTRCV.STATUS >= 16#80A1 AND #bMQTT_Connected THEN
       #bTCP_Connected := FALSE;
       #bMQTT_Connected := FALSE;

       IF #iErrIndex > 10 THEN
           #iErrIndex := 1;
       END_IF;

       #iErrIndex := #iErrIndex + 1;

       //Reinit all subscribed topics
       FOR #i := 1 TO 20 BY 1 DO
           "dbMQTT_MessageBuffer".IncomingMessages.Message[#i].iStatus := 0;
       END_FOR;

       #iStatePublish := #ciPubError;
   END_IF;

   #fbTCON(REQ := (#iStatePublish = #ciEstablishTCP),
           ID := #TCON_Param.ID,
           CONNECT := #TCON_Param);

   #fbTDISCON(REQ := (#iStatePublish = #ciPubError) ,
              ID := #TCON_Param.ID);

   #fbTSEND(REQ := (#iStatePublish = #ciPubConnectSend) OR (#iStatePublish = #ciPubSend) OR (#iStateSubscribe = #ciSubSendSubscribe) OR (#iStateSubscribe = #ciSubSendPubAck),
            ID := #TCON_Param.ID,
            LEN := #uiSendLen,
            DATA := #byData);

   //always listen after MQTT connected

   #fbTRCV(EN_R := (#bMQTT_Connected OR (#iStatePublish = #ciPubWaitConnack) OR (#iStatePublish = #ciPubWaitPubAck)),
           ID := #TCON_Param.ID,
           LEN := 1,
           DATA := #byData);

   #TON_ReceiveDataComplete(IN := NOT #fbTRCV.NDR,
                            PT := T#300ms);



   //Only receive 1 byte at a time. After 3 seconds of no data, message is considered complete.
   IF (#fbTRCV.NDR AND NOT #bConAckReceived AND NOT #bPubAckReceived AND NOT #bSubAckReceived AND NOT #bPublishReceived AND NOT #bReceiveMessageComplete) THEN

       #byDataNewMessage[#iNewDataIndex] := #byData[1];
       //check if we can calculate the total length of the message

       IF #iNewDataIndex >= 2 AND (#byDataNewMessage[#iNewDataIndex] AND 128) = 0 AND #iReceiveMessageLength = 0 THEN
           #iReceiveLengthCalcIndex := 2;
           #iLen := 0;
           #multiplier := 1;
           REPEAT

               #byTemp := #byDataNewMessage[#iReceiveLengthCalcIndex];
               #iLen := #iLen + (#byTemp AND 127) * #multiplier;
               #multiplier := #multiplier * 128;
               //TODO implement exception for length error
               #iReceiveLengthCalcIndex := #iReceiveLengthCalcIndex + 1;
           UNTIL ((#byTemp AND 128) = 0) END_REPEAT;
           #iReceiveMessageLength := #iLen;

       END_IF;
       IF (#iReceiveMessageLength + #iReceiveLengthCalcIndex - 1) = #iNewDataIndex THEN
           #bReceiveMessageComplete := TRUE;
       END_IF;
       #iNewDataIndex := #iNewDataIndex + 1;

   END_IF;

   //**********************************************************************************************************************
   // Reset all errors
   IF #bInResetError THEN
       #ERROR_MQTT.ConSendErr := FALSE;
       #ERROR_MQTT.ConSendTO := FALSE;
       #ERROR_MQTT.ConAckRcvErr := FALSE;
       #ERROR_MQTT.ConAckTO := FALSE;
       #ERROR_MQTT.ConAckIncReply := FALSE;
       #ERROR_MQTT.ConAckIncLen := FALSE;
       #ERROR_MQTT.ConAckUnacProt := FALSE;
       #ERROR_MQTT.ConAckIdRej := FALSE;
       #ERROR_MQTT.ConAckSerUn := FALSE;
       #ERROR_MQTT.ConAckUserPass := FALSE;
       #ERROR_MQTT.ConAckNotAut := FALSE;
       #ERROR_MQTT.ConAckUnknown := FALSE;
       #ERROR_MQTT.PubSendErr := FALSE;
       #ERROR_MQTT.PubSendTO := FALSE;
       #ERROR_MQTT.PubAckRcvErr := FALSE;
       #ERROR_MQTT.PubAckTO := FALSE;
       #ERROR_MQTT.PubAckIncReply := FALSE;
       #ERROR_MQTT.PubAckIncLen := FALSE;
       #ERROR_MQTT.PubAckPacketID := FALSE;
       #ERROR_MQTT.TcpErr := FALSE;
       #ERROR_MQTT.TcpTO := FALSE;
       #ERROR_MQTT.QueueOverflow := FALSE;
   END_IF;

   // At least one erorr is active - set output error flag
   #bOutError :=
   #ERROR_MQTT.ConSendErr OR
   #ERROR_MQTT.ConSendTO OR
   #ERROR_MQTT.ConAckRcvErr OR
   #ERROR_MQTT.ConAckTO OR
   #ERROR_MQTT.ConAckIncReply OR
   #ERROR_MQTT.ConAckIncLen OR
   #ERROR_MQTT.ConAckUnacProt OR
   #ERROR_MQTT.ConAckIdRej OR
   #ERROR_MQTT.ConAckSerUn OR
   #ERROR_MQTT.ConAckUserPass OR
   #ERROR_MQTT.ConAckNotAut OR
   #ERROR_MQTT.ConAckUnknown OR
   #ERROR_MQTT.PubSendErr OR
   #ERROR_MQTT.PubSendTO OR
   #ERROR_MQTT.PubAckRcvErr OR
   #ERROR_MQTT.PubAckTO OR
   #ERROR_MQTT.PubAckIncReply OR
   #ERROR_MQTT.PubAckIncLen OR
   #ERROR_MQTT.PubAckPacketID OR
   #ERROR_MQTT.SubSendErr OR
   #ERROR_MQTT.SubSendTimeout OR
   #ERROR_MQTT.SubAckIncReply OR
   #ERROR_MQTT.SubAckPacketID OR
   #ERROR_MQTT.SubAckRcvErr OR
   #ERROR_MQTT.SubAckTO OR
   #ERROR_MQTT.SubTopicNotFound OR
   #ERROR_MQTT.SubSendPubAckErr OR
   #ERROR_MQTT.SubSendPubAckTO OR
   #ERROR_MQTT.TcpErr OR
   #ERROR_MQTT.TcpTO OR
   #ERROR_MQTT.QueueOverflow;

   ENO := TRUE;
END_FUNCTION_BLOCK

FUNCTION "fcMQTT_SerializeMessage" : Void   // FC3, SCL
{ S7_Optimized_Access := 'TRUE' }
VERSION : 0.1
   VAR_INPUT
      sInTopic : String;   // Topic to push data to
      sInSerial : String;
      iInQoS : Int;   // Quality of Service needed
      Message : Variant;   // Data to be sent
   END_VAR
   VAR_OUTPUT
      bOutMessageSerialized : Bool;   // Set for one scan when message successfully entered into buffer
   END_VAR
   VAR_TEMP
      iTemp : Int;
      sTopicTemp1 : String;
      sTopicTemp2 : String;
      sTopicFull : String;
   END_VAR
   VAR CONSTANT
      sTopicPart1 : String := 'dev/';
      sTopicPart2 : String := '/msg/';
   END_VAR
BEGIN
   // Create Full Topic
   #sTopicTemp1 := CONCAT_STRING(IN1 := #sTopicPart1, IN2 := #sInSerial);
   #sTopicTemp2 := CONCAT_STRING(IN1 := #sTopicTemp1, IN2 := #sTopicPart2);
   #sTopicFull := CONCAT_STRING(IN1 := #sTopicTemp2, IN2 := #sInTopic);

   // Generate new global index to write    
   "dbMQTT_MessageBuffer".OutgoingMessages.iIndexWrite := "dbMQTT_MessageBuffer".OutgoingMessages.iIndexWrite + 1;
   // Check queue index at the end of the queue
   IF ("dbMQTT_MessageBuffer".OutgoingMessages.iIndexWrite > "dbMQTT_MessageBuffer".OutgoingMessages.iIndexMax) OR ("dbMQTT_MessageBuffer".OutgoingMessages.iIndexWrite <= 0) THEN
       "dbMQTT_MessageBuffer".OutgoingMessages.iIndexWrite := 1;
   END_IF;

   IF "dbMQTT_MessageBuffer".OutgoingMessages.Message["dbMQTT_MessageBuffer".OutgoingMessages.iIndexWrite].iStatus <> 0 THEN
       // Queue overfill detected
       "dbMQTT_MessageBuffer".OutgoingMessages.bErrorOverfill := true;
       #bOutMessageSerialized := FALSE;
   ELSE
       // Assing element to the queue
       // TODO: BLKMOV instead?
       "dbMQTT_MessageBuffer".OutgoingMessages.Message["dbMQTT_MessageBuffer".OutgoingMessages.iIndexWrite].sTopic := #sTopicFull;
       "dbMQTT_MessageBuffer".OutgoingMessages.Message["dbMQTT_MessageBuffer".OutgoingMessages.iIndexWrite].iQoS := #iInQoS;

       "dbMQTT_MessageBuffer".OutgoingMessages.Message["dbMQTT_MessageBuffer".OutgoingMessages.iIndexWrite].iMessageLength := 0;

       #iTemp := Serialize(SRC_VARIABLE := #Message, DEST_ARRAY => "dbMQTT_MessageBuffer".OutgoingMessages.Message["dbMQTT_MessageBuffer".OutgoingMessages.iIndexWrite].byValue,
                           POS := "dbMQTT_MessageBuffer".OutgoingMessages.Message["dbMQTT_MessageBuffer".OutgoingMessages.iIndexWrite].iMessageLength);

       // Update MQTT status
       "dbMQTT_MessageBuffer".OutgoingMessages.Message["dbMQTT_MessageBuffer".OutgoingMessages.iIndexWrite].iStatus := 10;

       #bOutMessageSerialized := TRUE;
   END_IF;

   ENO := TRUE;
END_FUNCTION

FUNCTION "fcMQTT_DeserializeMessageSubscribe" : Void   // FC5, SCL
{ S7_Optimized_Access := 'TRUE' }
VERSION : 0.1
   VAR_INPUT
      sInTopic : String;
      iInQoS : Int;
      iInBufferIndex : Int;
      sInSerial : String;
   END_VAR
   VAR_OUTPUT
      Message : Variant;
      bOutNewMessage : Bool;   // New message received, only active for one scan
   END_VAR
   VAR_TEMP
      iTemp : Int;
      iTemp2 : Int;
      diTemp : DInt;
      sTopicFull : String[75];
      sTopicTemp1 : String[16];
      sTopicTemp2 : String[21];
   END_VAR
   VAR CONSTANT
      sTopicPart1 : String := 'dev/';
      sTopicPart2 : String := '/cmd/';
   END_VAR
BEGIN
   // Create Full Topic
   #sTopicTemp1 := CONCAT_STRING(IN1 := #sTopicPart1, IN2 := #sInSerial);
   #sTopicTemp2 := CONCAT_STRING(IN1 := #sTopicTemp1, IN2 := #sTopicPart2);
   #sTopicFull := CONCAT_STRING(IN1 := #sTopicTemp2, IN2 := #sInTopic);


   //Check if subscribed

   IF ("dbMQTT_MessageBuffer".IncomingMessages.Message[#iInBufferIndex].iStatus = "ciSubDisabled") THEN
       "dbMQTT_MessageBuffer".IncomingMessages.Message[#iInBufferIndex].iStatus := "ciSubReadyToSub";
       "dbMQTT_MessageBuffer".IncomingMessages.Message[#iInBufferIndex].sTopic := #sTopicFull;
       "dbMQTT_MessageBuffer".IncomingMessages.Message[#iInBufferIndex].iQoS := #iInQoS;
   END_IF;

   IF ("dbMQTT_MessageBuffer".IncomingMessages.Message[#iInBufferIndex].iStatus = "ciSubMessageReceived") THEN
       #diTemp := 0;
       #iTemp := Deserialize(SRC_ARRAY := "dbMQTT_MessageBuffer".IncomingMessages.Message[#iInBufferIndex].byValue, DEST_VARIABLE => #Message, POS := #diTemp);
       "dbMQTT_MessageBuffer".IncomingMessages.Message[#iInBufferIndex].iStatus := "ciSubSubscribed";
       #bOutNewMessage := true;
   END_IF;
END_FUNCTION

// ===== library: MasterCopy "dbMessages" =====

DATA_BLOCK "dbMessages"   // DB1
{ S7_Optimized_Access := 'TRUE' }
VERSION : 0.1
   VAR
      SendData : Struct
         iInt : Int;
         rReal : Real;
      END_STRUCT;
      RecieveData : Struct
         bMessage : Bool;
         diDint : DInt;
      END_STRUCT;
   END_VAR
BEGIN
END_DATA_BLOCK

// ===== library: MasterCopy "dbMQTT_MessageBuffer" =====

DATA_BLOCK "dbMQTT_MessageBuffer"   // DB35
{ S7_Optimized_Access := 'FALSE' }
VERSION : 0.1
   VAR
      OutgoingMessages : "udtMQTT_PublishMessageBuffer";
      IncomingMessages : "udtMQTT_SubcribeMessageBuffer";
   END_VAR
BEGIN
   OutgoingMessages.iIndexMax := 3;
END_DATA_BLOCK

// ===== library: MasterCopy "IOT Communication" =====

FUNCTION_BLOCK "IOT Communication"   // FB18, SCL
{ S7_Optimized_Access := 'TRUE' }
VERSION : 0.1
   VAR
      MQTT : "fbMQTT_V2";
      MqttError : "udtError_MQTT";
      TCON_MQTT : TCON_Param;
      bMessageSerialized : Bool;
      bMessageReceived : Bool;
   END_VAR
   VAR_TEMP
      bTemp : Bool;
   END_VAR
   VAR CONSTANT
      siId : String := 'UniqueId';
   END_VAR
BEGIN
   // MQTT communication control driver
   #MQTT(sInClientID := 'Client ID',
                sInUserName := 'Serial Number', //Typically used to create unique login
                sInPassword := 'Password',
                bInResetError:=#bTemp,
                ERROR_MQTT := #MqttError,
                TCON_Param := #TCON_MQTT);

   "fcMQTT_SerializeMessage"(sInTopic := 'FirstScan',
                             sInSerial := #siId, //Appended in the function to make the topic unique
                             iInQoS := 0,
                             Message := "dbMessages".SendData,
                             bOutMessageSerialized => #bMessageSerialized);

   // Monitor IOT for new data
   "fcMQTT_DeserializeMessageSubscribe"(sInTopic := 'TopicName',
                                        iInQoS := 0,
                                        iInBufferIndex := 0,
                                        sInSerial := #siId, //Appended to topic name to create unique topic
                                        Message => "dbMessages".RecieveData,
                                        bOutNewMessage => #bMessageReceived);
END_FUNCTION_BLOCK

// ===== library: MasterCopy "IOT Constants" =====

VAR_GLOBAL CONSTANT   // PLC tag table "IOT Constants"
   "ciDisablePublish" : Int := 0;
   "ciSubDisabled" : Int := 0;
   "ciSubReadyToSub" : Int := 10;
   "ciReadyToPublish" : Int := 10;
   "ciSubSubscribed" : Int := 20;
   "ciSubMessageReceived" : Int := 15;
END_VAR